# EPICS autosave request: iocBoot/ioc13MeasCompETC_3/auto_settings.req
file "ETC_settings.req", P=$(P)
